FUNCTION_BLOCK Sequence3
VAR_INPUT
END_VAR
VAR_OUTPUT
	bMoveError : BOOL;
	bSequenceError : BOOL;
END_VAR
VAR
	nState : INT;
	fbMoveVelocity: MC_MoveVelocity;
	fbHalt: MC_Halt;
	bHaltExecute: BOOL;
	bResetExecute: BOOL;
	bPowerExecute: BOOL;
	bVelocityExecute : BOOL;
	MC_MoveAbsolute1: MC_MoveAbsolute;
	MC_Stop1: MC_Stop;
END_VAR
VAR_IN_OUT
END_VAR

		(*fbHalt(
			Axis:= GVL_Conveyer.ConveyerAxis, 
			Execute:= bHaltExecute
			);*)
			
		fbMoveVelocity(
			Axis:= GVL_Conveyer.ConveyerAxis, 
			Execute:= bVelocityExecute, 
			Velocity:= 600, 
			Direction := MC_Negative_Direction
			);
		
		MC_Stop1(
			Axis:= GVL_Conveyer.ConveyerAxis, 
			Execute:= bHaltExecute);	
			
CASE nState OF
	
0: // Call velocity move
	IF NOT GVL_Conveyer.bSensor THEN
		bVelocityExecute := TRUE;
		nState := 1;
	END_IF
	
1: // Set vel move low
	IF (GVL_Conveyer.ConveyerAxis.NcToPlc.ActVelo > 1) OR (GVL_Conveyer.ConveyerAxis.NcToPlc.ActVelo < -1) THEN
		bVelocityExecute := FALSE;
		nState := 5;
	END_IF
	
5: // Call stop movement when something is there
	IF GVL_Conveyer.bSensor THEN
		GVL_Conveyer.bConveyerReadyToPick := TRUE;
		bHaltExecute := TRUE;
		nState := 10;
	END_IF
	
10: // Check if halt is complete
	IF MC_Stop1.Done THEN
		nState := 15;
		bHaltExecute := FALSE;
	END_IF
	
15: // If sensor low, then call ready to move high
	IF NOT GVL_Conveyer.bSensor AND GVL_conveyer.bConveyerReadyToMove THEN
		GVL_Conveyer.bConveyerReadyToPick := FALSE;
		
		nState := 0;
	END_IF
			
999:
	IF NOT fbMoveVelocity.Error AND NOT fbHalt.Error THEN
		
		nState := 0;
		bSequenceError := FALSE;
	ELSE
		bSequenceError := TRUE;
	END_IF
END_CASE

END_FUNCTION_BLOCK

(* stored: Version 1.1.0.1, ProductVersion 3.1.4024.11
   POU Sequence3: Id {e15a6fb5-808f-4738-8ea3-952c583c643e}, SpecialFunc None *)
